// TIA Portal V20 export
// export: Created 2025-12-01T14:56:59.4863096Z, ExportSetting None, DisplayName Totally Integrated Automation Portal, DisplayVersion V20 Update 3, DisplayName TIA Portal Openness, DisplayVersion V20 Update 3, DisplayName TIA Portal Version Control Interface, DisplayVersion V20 Update 3, DisplayName STEP 7 Professional, DisplayVersion V20 Update 3, DisplayName STEP 7 Safety, DisplayVersion V20 Update 2, DisplayName WinCC Basic/Comfort/Advanced, DisplayVersion V20 Update 3, DisplayName WinCC Professional, DisplayVersion V20 Update 3, DisplayName WinCC Unified, DisplayVersion V20 Update 3
FUNCTION "FC415_DesvioPosicionPaletizado" : Void   // FC415, LAD
{ S7_Optimized_Access := 'FALSE' }
NAME : 20180830
VERSION : 1.0
// stored: AutoNumber false, SetENOAutomatically false
   VAR_INPUT
      NumeroMesa : UInt;
      Pos_Der_Act : Bool;
      Pos_Der_Desact : Bool;
      Pos_Izda_Act : Bool;
      Pos_Izda_Desact : Bool;
      V_TimeOut : UDInt;   // en milisegundos
      V_Reposo : UDInt;   // en milisegundos
   END_VAR
   VAR_TEMP
      InformeDatosUT : "UDT_Informe_DatosUT";
      Ir_Derecha : Bool;
      Ir_Izda : Bool;
      Ir_Centro : Bool;
      Sin_UT : Bool;
      Errormovimiento : Bool;
      ReposoOK : Bool;
   END_VAR
   VAR_TEMP   // added for the SCL form of the ladder/FBD networks
      _w1 : Bool;
   END_VAR
BEGIN

REGION Network 1: Extraer Información
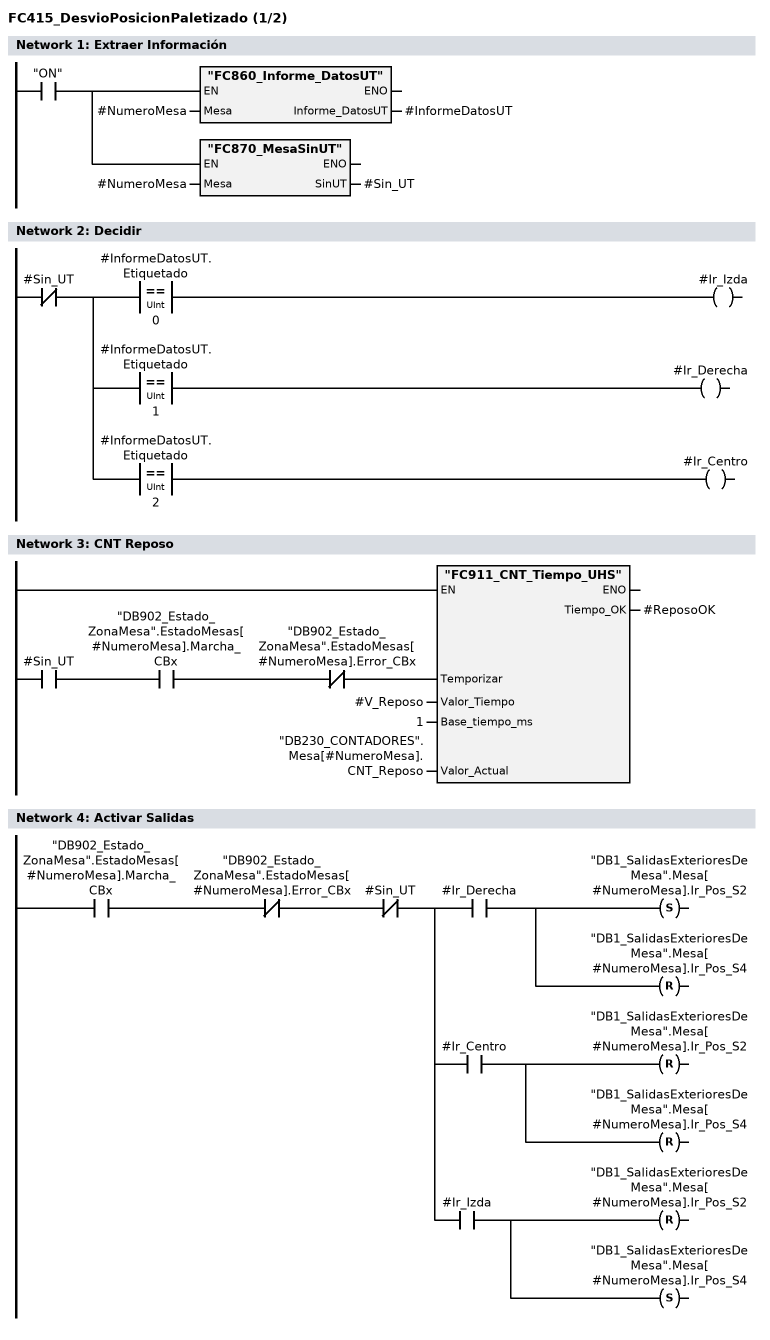
   RUNG wire#powerrail
      Contact( "ON" )
      wire#w1
      "FC860_Informe_DatosUT"(Mesa := #NumeroMesa, Informe_DatosUT => #InformeDatosUT)
   END_RUNG
   RUNG wire#w1
      "FC870_MesaSinUT"(Mesa := #NumeroMesa, SinUT => #Sin_UT)
   END_RUNG
   // the same network as SCL:
   #_w1 := "ON";
   IF #_w1 THEN
       "FC860_Informe_DatosUT"(Mesa := #NumeroMesa, Informe_DatosUT => #InformeDatosUT);
       "FC870_MesaSinUT"(Mesa := #NumeroMesa, SinUT => #Sin_UT);
   END_IF;
END_REGION

REGION Network 2: Decidir
   RUNG wire#powerrail
      I_Contact( #Sin_UT )
      wire#w1
      { S7_Templates := "SrcType := UInt" } EQ_Contact(in1 := #InformeDatosUT.Etiquetado, in2 := 0)
      Coil( #Ir_Izda )
   END_RUNG
   RUNG wire#w1
      { S7_Templates := "SrcType := UInt" } EQ_Contact(in1 := #InformeDatosUT.Etiquetado, in2 := 1)
      Coil( #Ir_Derecha )
   END_RUNG
   RUNG wire#w1
      { S7_Templates := "SrcType := UInt" } EQ_Contact(in1 := #InformeDatosUT.Etiquetado, in2 := 2)
      Coil( #Ir_Centro )
   END_RUNG
   // the same network as SCL:
   #Ir_Izda := NOT #Sin_UT AND (#InformeDatosUT.Etiquetado = 0);
   #Ir_Derecha := NOT #Sin_UT AND (#InformeDatosUT.Etiquetado = 1);
   #Ir_Centro := NOT #Sin_UT AND (#InformeDatosUT.Etiquetado = 2);
END_REGION

REGION Network 3: CNT Reposo
   RUNG wire#powerrail
      "FC911_CNT_Tiempo_UHS"(Temporizar := wire#w1, Valor_Tiempo := #V_Reposo, Base_tiempo_ms := 1, Valor_Actual := "DB230_CONTADORES".Mesa[#NumeroMesa].CNT_Reposo, Tiempo_OK => #ReposoOK)
   END_RUNG
   RUNG wire#powerrail
      Contact( #Sin_UT )
      Contact( "DB902_Estado_ZonaMesa".EstadoMesas[#NumeroMesa].Marcha_CBx )
      I_Contact( "DB902_Estado_ZonaMesa".EstadoMesas[#NumeroMesa].Error_CBx )
   END_RUNG wire#w1
   // the same network as SCL:
   "FC911_CNT_Tiempo_UHS"(Temporizar := #Sin_UT AND "DB902_Estado_ZonaMesa".EstadoMesas[#NumeroMesa].Marcha_CBx AND NOT "DB902_Estado_ZonaMesa".EstadoMesas[#NumeroMesa].Error_CBx,
                          Valor_Tiempo := #V_Reposo,
                          Base_tiempo_ms := 1,
                          Valor_Actual := "DB230_CONTADORES".Mesa[#NumeroMesa].CNT_Reposo,
                          Tiempo_OK => #ReposoOK);
END_REGION

REGION Network 4: Activar Salidas
   RUNG wire#powerrail
      Contact( "DB902_Estado_ZonaMesa".EstadoMesas[#NumeroMesa].Marcha_CBx )
      I_Contact( "DB902_Estado_ZonaMesa".EstadoMesas[#NumeroMesa].Error_CBx )
      I_Contact( #Sin_UT )
      wire#w1
      Contact( #Ir_Derecha )
      wire#w2
      S_Coil( "DB1_SalidasExterioresDeMesa".Mesa[#NumeroMesa].Ir_Pos_S2 )
   END_RUNG
   RUNG wire#w2
      R_Coil( "DB1_SalidasExterioresDeMesa".Mesa[#NumeroMesa].Ir_Pos_S4 )
   END_RUNG
   RUNG wire#w1
      Contact( #Ir_Centro )
      wire#w3
      R_Coil( "DB1_SalidasExterioresDeMesa".Mesa[#NumeroMesa].Ir_Pos_S2 )
   END_RUNG
   RUNG wire#w3
      R_Coil( "DB1_SalidasExterioresDeMesa".Mesa[#NumeroMesa].Ir_Pos_S4 )
   END_RUNG
   RUNG wire#w1
      Contact( #Ir_Izda )
      wire#w4
      R_Coil( "DB1_SalidasExterioresDeMesa".Mesa[#NumeroMesa].Ir_Pos_S2 )
   END_RUNG
   RUNG wire#w4
      S_Coil( "DB1_SalidasExterioresDeMesa".Mesa[#NumeroMesa].Ir_Pos_S4 )
   END_RUNG
   // the same network as SCL:
   #_w1 := "DB902_Estado_ZonaMesa".EstadoMesas[#NumeroMesa].Marcha_CBx AND NOT "DB902_Estado_ZonaMesa".EstadoMesas[#NumeroMesa].Error_CBx AND NOT #Sin_UT;
   IF #_w1 AND #Ir_Derecha THEN
       "DB1_SalidasExterioresDeMesa".Mesa[#NumeroMesa].Ir_Pos_S2 := TRUE;
       "DB1_SalidasExterioresDeMesa".Mesa[#NumeroMesa].Ir_Pos_S4 := FALSE;
   END_IF;
   IF #_w1 AND #Ir_Centro THEN
       "DB1_SalidasExterioresDeMesa".Mesa[#NumeroMesa].Ir_Pos_S2 := FALSE;
       "DB1_SalidasExterioresDeMesa".Mesa[#NumeroMesa].Ir_Pos_S4 := FALSE;
   END_IF;
   IF #_w1 AND #Ir_Izda THEN
       "DB1_SalidasExterioresDeMesa".Mesa[#NumeroMesa].Ir_Pos_S2 := FALSE;
       "DB1_SalidasExterioresDeMesa".Mesa[#NumeroMesa].Ir_Pos_S4 := TRUE;
   END_IF;
END_REGION

REGION Network 5: ---
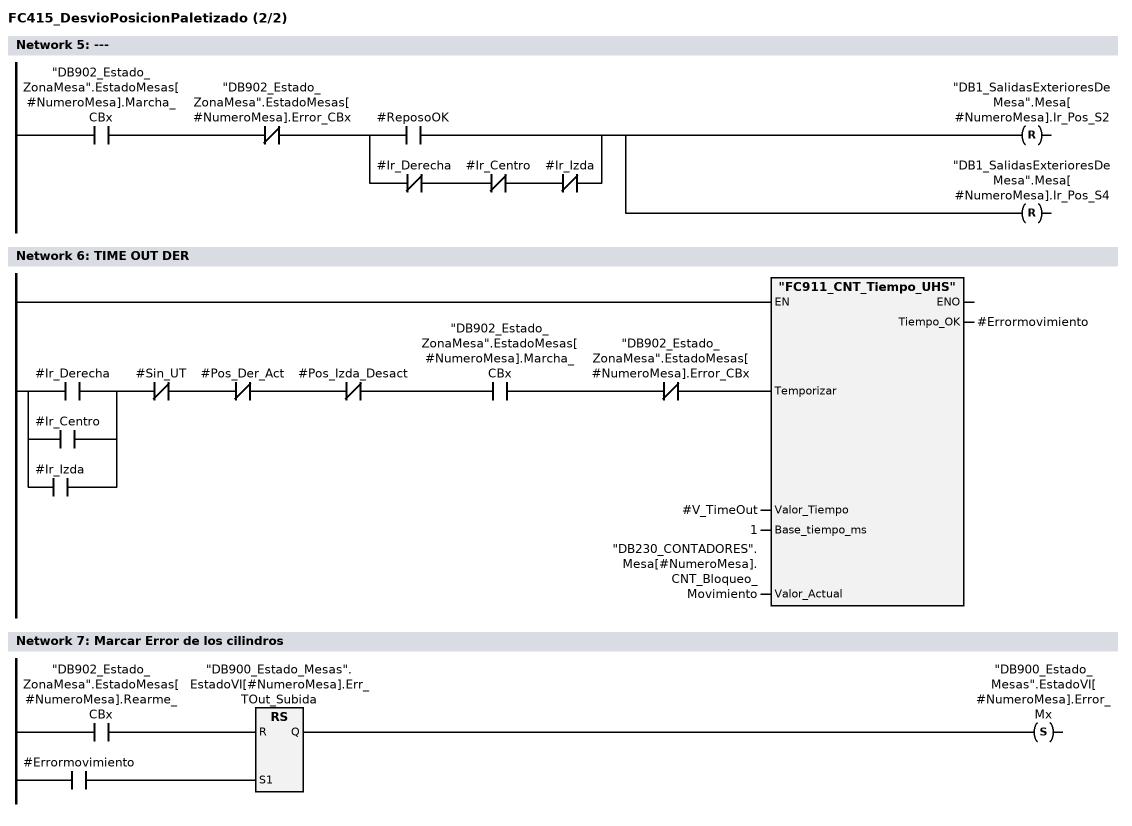
   RUNG wire#powerrail
      Contact( "DB902_Estado_ZonaMesa".EstadoMesas[#NumeroMesa].Marcha_CBx )
      I_Contact( "DB902_Estado_ZonaMesa".EstadoMesas[#NumeroMesa].Error_CBx )
      wire#w1
      Contact( #ReposoOK )
      wire#w2
      R_Coil( "DB1_SalidasExterioresDeMesa".Mesa[#NumeroMesa].Ir_Pos_S2 )
   END_RUNG
   RUNG wire#w1
      I_Contact( #Ir_Derecha )
      I_Contact( #Ir_Centro )
      I_Contact( #Ir_Izda )
   END_RUNG wire#w2
   RUNG wire#w2
      R_Coil( "DB1_SalidasExterioresDeMesa".Mesa[#NumeroMesa].Ir_Pos_S4 )
   END_RUNG
   // the same network as SCL:
   #_w1 := "DB902_Estado_ZonaMesa".EstadoMesas[#NumeroMesa].Marcha_CBx AND NOT "DB902_Estado_ZonaMesa".EstadoMesas[#NumeroMesa].Error_CBx AND (#ReposoOK OR (NOT #Ir_Derecha AND NOT #Ir_Centro AND NOT #Ir_Izda));
   IF #_w1 THEN
       "DB1_SalidasExterioresDeMesa".Mesa[#NumeroMesa].Ir_Pos_S2 := FALSE;
       "DB1_SalidasExterioresDeMesa".Mesa[#NumeroMesa].Ir_Pos_S4 := FALSE;
   END_IF;
END_REGION

REGION Network 6: TIME OUT DER
   RUNG wire#powerrail
      "FC911_CNT_Tiempo_UHS"(Temporizar := wire#w2, Valor_Tiempo := #V_TimeOut, Base_tiempo_ms := 1, Valor_Actual := "DB230_CONTADORES".Mesa[#NumeroMesa].CNT_Bloqueo_Movimiento, Tiempo_OK => #Errormovimiento)
   END_RUNG
   RUNG wire#powerrail
      Contact( #Ir_Derecha )
      wire#w1
      I_Contact( #Sin_UT )
      I_Contact( #Pos_Der_Act )
      I_Contact( #Pos_Izda_Desact )
      Contact( "DB902_Estado_ZonaMesa".EstadoMesas[#NumeroMesa].Marcha_CBx )
      I_Contact( "DB902_Estado_ZonaMesa".EstadoMesas[#NumeroMesa].Error_CBx )
   END_RUNG wire#w2
   RUNG wire#powerrail
      Contact( #Ir_Centro )
   END_RUNG wire#w1
   RUNG wire#powerrail
      Contact( #Ir_Izda )
   END_RUNG wire#w1
   // the same network as SCL:
   "FC911_CNT_Tiempo_UHS"(Temporizar := (#Ir_Derecha OR #Ir_Centro OR #Ir_Izda) AND NOT #Sin_UT AND NOT #Pos_Der_Act AND NOT #Pos_Izda_Desact AND "DB902_Estado_ZonaMesa".EstadoMesas[#NumeroMesa].Marcha_CBx AND NOT "DB902_Estado_ZonaMesa".EstadoMesas[#NumeroMesa].Error_CBx,
                          Valor_Tiempo := #V_TimeOut,
                          Base_tiempo_ms := 1,
                          Valor_Actual := "DB230_CONTADORES".Mesa[#NumeroMesa].CNT_Bloqueo_Movimiento,
                          Tiempo_OK => #Errormovimiento);
END_REGION

REGION Network 7: Marcar Error de los cilindros
   RUNG wire#powerrail
      Contact( "DB902_Estado_ZonaMesa".EstadoMesas[#NumeroMesa].Rearme_CBx )
      S_RS(operand := "DB900_Estado_Mesas".EstadoVI[#NumeroMesa].Err_TOut_Subida, s1 := wire#w1)
      S_Coil( "DB900_Estado_Mesas".EstadoVI[#NumeroMesa].Error_Mx )
   END_RUNG
   RUNG wire#powerrail
      Contact( #Errormovimiento )
   END_RUNG wire#w1
   // the same network as SCL:
   IF "DB902_Estado_ZonaMesa".EstadoMesas[#NumeroMesa].Rearme_CBx THEN
       "DB900_Estado_Mesas".EstadoVI[#NumeroMesa].Err_TOut_Subida := FALSE;   // RS flip-flop
   END_IF;
   IF #Errormovimiento THEN "DB900_Estado_Mesas".EstadoVI[#NumeroMesa].Err_TOut_Subida := TRUE; END_IF;
   IF "DB900_Estado_Mesas".EstadoVI[#NumeroMesa].Err_TOut_Subida THEN
       "DB900_Estado_Mesas".EstadoVI[#NumeroMesa].Error_Mx := TRUE;
   END_IF;
END_REGION
END_FUNCTION
